KUKA KRL program: Milling_8_2.src

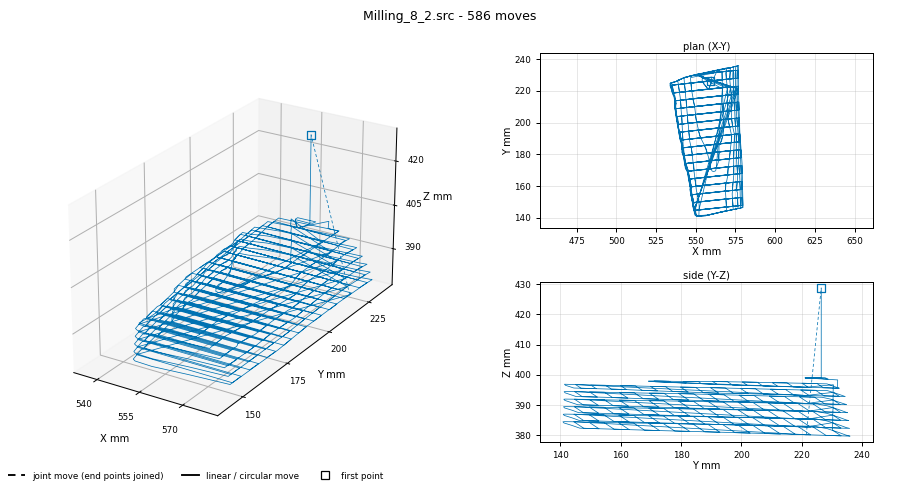
[picture p0: tool path of Milling_8_2.src, 586 of 588 moves have a stored position in this frame; points joined in program order, loops and branches not executed]
&ACCESS RVP
&REL 1
&PARAM TEMPLATE = C:\KRC\Roboter\Template\vorgabe
&PARAM EDITMASK = *
DEF Milling_8_2 ( )


;FOLD INI
;FOLD BASISTECH INI
GLOBAL INTERRUPT DECL 3 WHEN $STOPMESS==TRUE DO IR_STOPM ( )
INTERRUPT ON 3
BAS (#INITMOV,0 )
;ENDFOLD (BASISTECH INI)
;ENDFOLD (INI)

;FOLD STARTPOSITION - BASE IS 0, TOOL IS 5, SPEED IS 15%, POSITION IS A1 5,A2 -90,A3 100,A4 5,A5 -10,A6 -5,E1 0,E2 0,E3 0,E4 0
$BWDSTART = FALSE
PDAT_ACT = {VEL 15,ACC 100,APO_DIST 50}
FDAT_ACT = {TOOL_NO 5,BASE_NO 0,IPO_FRAME #BASE}
BAS (#PTP_PARAMS,15)
PTP  {A1 5,A2 -90,A3 100,A4 5,A5 -10,A6 -5,E1 0,E2 0,E3 0,E4 0}
;ENDFOLD

;FOLD LIN SPEED IS 0.1 m/sec, INTERPOLATION SETTINGS IN FOLD
$VEL.CP=0.1
$ADVANCE=3
;ENDFOLD

BAS(#VEL_PTP,2)
PTP {X 559.273, Y 226.42, Z 428.722, A -154.581, B 85.803, C -170.798, E1 0, E2 0, E3 0, E4 0, S 'B010'}
$VEL.CP=0.012
LIN {X 559.273, Y 226.42, Z 398.722, A -154.581, B 85.803, C -170.798, E1 0, E2 0, E3 0, E4 0}
LIN {X 554.276, Y 225.886, Z 399.07, A -154.581, B 85.803, C -170.798, E1 0, E2 0, E3 0, E4 0}
LIN {X 557.594, Y 221.214, Z 398.997, A -154.581, B 85.803, C -170.798, E1 0, E2 0, E3 0, E4 0}
LIN {X 558.179, Y 221.276, Z 398.957, A -154.581, B 85.803, C -170.798, E1 0, E2 0, E3 0, E4 0}
LIN {X 558.124, Y 221.152, Z 398.964, A -154.581, B 85.803, C -170.798, E1 0, E2 0, E3 0, E4 0}
LIN {X 559.233, Y 224.054, Z 398.799, A -154.581, B 85.803, C -170.798, E1 0, E2 0, E3 0, E4 0}
LIN {X 559.279, Y 226.805, Z 398.71, A -154.581, B 85.803, C -170.798, E1 0, E2 0, E3 0, E4 0}
LIN {X 559.896, Y 227.132, Z 398.659, A -154.581, B 85.803, C -170.798, E1 0, E2 0, E3 0, E4 0}
LIN {X 560.102, Y 228.698, Z 398.595, A -154.581, B 85.803, C -170.798, E1 0, E2 0, E3 0, E4 0}
LIN {X 554.041, Y 227.675, Z 399.029, A -154.581, B 85.803, C -170.798, E1 0, E2 0, E3 0, E4 0}
LIN {X 554.023, Y 226.451, Z 399.069, A -154.581, B 85.803, C -170.798, E1 0, E2 0, E3 0, E4 0}
LIN {X 555.02, Y 224.234, Z 399.073, A -154.581, B 85.803, C -170.798, E1 0, E2 0, E3 0, E4 0}
LIN {X 557.587, Y 221.412, Z 398.992, A -154.581, B 85.803, C -170.798, E1 0, E2 0, E3 0, E4 0}
LIN {X 557.599, Y 221.063, Z 399.002, A -154.581, B 85.803, C -170.798, E1 0, E2 0, E3 0, E4 0}
LIN {X 557.929, Y 221.029, Z 398.981, A -154.581, B 85.803, C -170.798, E1 0, E2 0, E3 0, E4 0}
LIN {X 558.124, Y 221.152, Z 398.964, A -154.581, B 85.803, C -170.798, E1 0, E2 0, E3 0, E4 0}
LIN {X 563.082, Y 231.869, Z 398.3, A -154.581, B 85.803, C -170.798, E1 0, E2 0, E3 0, E4 0}
LIN {X 562.917, Y 231.79, Z 395.806, A -154.581, B 85.803, C -170.798, E1 0, E2 0, E3 0, E4 0}
LIN {X 566.518, Y 232.175, Z 395.555, A -154.581, B 85.803, C -170.798, E1 0, E2 0, E3 0, E4 0}
LIN {X 566.596, Y 227.157, Z 395.708, A -154.581, B 85.803, C -170.798, E1 0, E2 0, E3 0, E4 0}
LIN {X 546.975, Y 225.06, Z 397.075, A -154.581, B 85.803, C -170.798, E1 0, E2 0, E3 0, E4 0}
LIN {X 547.397, Y 220.078, Z 397.204, A -154.581, B 85.803, C -170.798, E1 0, E2 0, E3 0, E4 0}
LIN {X 566.723, Y 222.143, Z 395.858, A -154.581, B 85.803, C -170.798, E1 0, E2 0, E3 0, E4 0}
LIN {X 566.992, Y 217.145, Z 395.997, A -154.581, B 85.803, C -170.798, E1 0, E2 0, E3 0, E4 0}
LIN {X 548.065, Y 215.122, Z 397.316, A -154.581, B 85.803, C -170.798, E1 0, E2 0, E3 0, E4 0}
LIN {X 549.244, Y 210.221, Z 397.392, A -154.581, B 85.803, C -170.798, E1 0, E2 0, E3 0, E4 0}
LIN {X 567.155, Y 212.135, Z 396.144, A -154.581, B 85.803, C -170.798, E1 0, E2 0, E3 0, E4 0}
LIN {X 567.374, Y 207.131, Z 396.288, A -154.581, B 85.803, C -170.798, E1 0, E2 0, E3 0, E4 0}
LIN {X 549.724, Y 205.245, Z 397.517, A -154.581, B 85.803, C -170.798, E1 0, E2 0, E3 0, E4 0}
LIN {X 550.455, Y 200.296, Z 397.624, A -154.581, B 85.803, C -170.798, E1 0, E2 0, E3 0, E4 0}
LIN {X 567.339, Y 202.101, Z 396.448, A -154.581, B 85.803, C -170.798, E1 0, E2 0, E3 0, E4 0}
LIN {X 567.528, Y 197.094, Z 396.594, A -154.581, B 85.803, C -170.798, E1 0, E2 0, E3 0, E4 0}
LIN {X 551.488, Y 195.379, Z 397.711, A -154.581, B 85.803, C -170.798, E1 0, E2 0, E3 0, E4 0}
LIN {X 553.074, Y 190.522, Z 397.758, A -154.581, B 85.803, C -170.798, E1 0, E2 0, E3 0, E4 0}
LIN {X 567.026, Y 192.013, Z 396.787, A -154.581, B 85.803, C -170.798, E1 0, E2 0, E3 0, E4 0}
LIN {X 565.372, Y 186.809, Z 397.06, A -154.581, B 85.803, C -170.798, E1 0, E2 0, E3 0, E4 0}
LIN {X 555.414, Y 185.745, Z 397.754, A -154.581, B 85.803, C -170.798, E1 0, E2 0, E3 0, E4 0}
LIN {X 557.158, Y 180.904, Z 397.791, A -154.581, B 85.803, C -170.798, E1 0, E2 0, E3 0, E4 0}
LIN {X 564.666, Y 181.706, Z 397.268, A -154.581, B 85.803, C -170.798, E1 0, E2 0, E3 0, E4 0}
LIN {X 564.615, Y 176.674, Z 397.43, A -154.581, B 85.803, C -170.798, E1 0, E2 0, E3 0, E4 0}
LIN {X 558.479, Y 176.018, Z 397.857, A -154.581, B 85.803, C -170.798, E1 0, E2 0, E3 0, E4 0}
LIN {X 559.339, Y 171.083, Z 397.956, A -154.581, B 85.803, C -170.798, E1 0, E2 0, E3 0, E4 0}
LIN {X 562.949, Y 171.469, Z 397.704, A -154.581, B 85.803, C -170.798, E1 0, E2 0, E3 0, E4 0}
LIN {X 566.751, Y 221.283, Z 395.883, A -154.581, B 85.803, C -170.798, E1 0, E2 0, E3 0, E4 0}
LIN {X 566.546, Y 229.177, Z 395.648, A -154.581, B 85.803, C -170.798, E1 0, E2 0, E3 0, E4 0}
LIN {X 566.512, Y 232.489, Z 395.546, A -154.581, B 85.803, C -170.798, E1 0, E2 0, E3 0, E4 0}
LIN {X 559.172, Y 230.807, Z 396.086, A -154.581, B 85.803, C -170.798, E1 0, E2 0, E3 0, E4 0}
LIN {X 546.627, Y 228.324, Z 396.995, A -154.581, B 85.803, C -170.798, E1 0, E2 0, E3 0, E4 0}
LIN {X 547.352, Y 220.421, Z 397.196, A -154.581, B 85.803, C -170.798, E1 0, E2 0, E3 0, E4 0}
LIN {X 549.239, Y 210.57, Z 397.381, A -154.581, B 85.803, C -170.798, E1 0, E2 0, E3 0, E4 0}
LIN {X 549.237, Y 210.401, Z 397.387, A -154.581, B 85.803, C -170.798, E1 0, E2 0, E3 0, E4 0}
LIN {X 550.242, Y 201.891, Z 397.588, A -154.581, B 85.803, C -170.798, E1 0, E2 0, E3 0, E4 0}
LIN {X 552.523, Y 191.514, Z 397.764, A -154.581, B 85.803, C -170.798, E1 0, E2 0, E3 0, E4 0}
LIN {X 556.467, Y 183.635, Z 397.751, A -154.581, B 85.803, C -170.798, E1 0, E2 0, E3 0, E4 0}
LIN {X 558.139, Y 177.602, Z 397.83, A -154.581, B 85.803, C -170.798, E1 0, E2 0, E3 0, E4 0}
LIN {X 558.213, Y 176.662, Z 397.854, A -154.581, B 85.803, C -170.798, E1 0, E2 0, E3 0, E4 0}
LIN {X 558.667, Y 175.563, Z 397.859, A -154.581, B 85.803, C -170.798, E1 0, E2 0, E3 0, E4 0}
LIN {X 558.417, Y 174.065, Z 397.923, A -154.581, B 85.803, C -170.798, E1 0, E2 0, E3 0, E4 0}
LIN {X 558.896, Y 172.014, Z 397.956, A -154.581, B 85.803, C -170.798, E1 0, E2 0, E3 0, E4 0}
LIN {X 560.318, Y 169.434, Z 397.943, A -154.581, B 85.803, C -170.798, E1 0, E2 0, E3 0, E4 0}
LIN {X 561.305, Y 169.205, Z 397.884, A -154.581, B 85.803, C -170.798, E1 0, E2 0, E3 0, E4 0}
LIN {X 562.277, Y 169.501, Z 397.811, A -154.581, B 85.803, C -170.798, E1 0, E2 0, E3 0, E4 0}
LIN {X 562.575, Y 169.872, Z 397.779, A -154.581, B 85.803, C -170.798, E1 0, E2 0, E3 0, E4 0}
LIN {X 562.981, Y 171.756, Z 397.693, A -154.581, B 85.803, C -170.798, E1 0, E2 0, E3 0, E4 0}
LIN {X 564.651, Y 176.325, Z 397.438, A -154.581, B 85.803, C -170.798, E1 0, E2 0, E3 0, E4 0}
LIN {X 564.581, Y 176.991, Z 397.422, A -154.581, B 85.803, C -170.798, E1 0, E2 0, E3 0, E4 0}
LIN {X 564.319, Y 177.275, Z 397.43, A -154.581, B 85.803, C -170.798, E1 0, E2 0, E3 0, E4 0}
LIN {X 564.116, Y 178.487, Z 397.406, A -154.581, B 85.803, C -170.798, E1 0, E2 0, E3 0, E4 0}
LIN {X 564.61, Y 180.491, Z 397.31, A -154.581, B 85.803, C -170.798, E1 0, E2 0, E3 0, E4 0}
LIN {X 564.637, Y 185.466, Z 397.151, A -154.581, B 85.803, C -170.798, E1 0, E2 0, E3 0, E4 0}
LIN {X 565, Y 186.057, Z 397.109, A -154.581, B 85.803, C -170.798, E1 0, E2 0, E3 0, E4 0}
LIN {X 565.01, Y 186.246, Z 397.102, A -154.581, B 85.803, C -170.798, E1 0, E2 0, E3 0, E4 0}
LIN {X 566.215, Y 188.326, Z 396.957, A -154.581, B 85.803, C -170.798, E1 0, E2 0, E3 0, E4 0}
LIN {X 567.259, Y 192.546, Z 396.755, A -154.581, B 85.803, C -170.798, E1 0, E2 0, E3 0, E4 0}
LIN {X 567.711, Y 198.434, Z 396.539, A -154.581, B 85.803, C -170.798, E1 0, E2 0, E3 0, E4 0}
LIN {X 567.365, Y 200.775, Z 396.488, A -154.581, B 85.803, C -170.798, E1 0, E2 0, E3 0, E4 0}
LIN {X 567.009, Y 210.951, Z 396.191, A -154.581, B 85.803, C -170.798, E1 0, E2 0, E3 0, E4 0}
LIN {X 567.109, Y 211.539, Z 396.166, A -154.581, B 85.803, C -170.798, E1 0, E2 0, E3 0, E4 0}
LIN {X 566.841, Y 217.785, Z 395.987, A -154.581, B 85.803, C -170.798, E1 0, E2 0, E3 0, E4 0}
LIN {X 566.751, Y 221.283, Z 395.883, A -154.581, B 85.803, C -170.798, E1 0, E2 0, E3 0, E4 0}
LIN {X 550.024, Y 230.427, Z 396.705, A -154.581, B 85.803, C -170.798, E1 0, E2 0, E3 0, E4 0}
LIN {X 549.859, Y 230.349, Z 394.212, A -154.581, B 85.803, C -170.798, E1 0, E2 0, E3 0, E4 0}
LIN {X 569.128, Y 232.408, Z 392.87, A -154.581, B 85.803, C -170.798, E1 0, E2 0, E3 0, E4 0}
LIN {X 569.258, Y 227.395, Z 393.019, A -154.581, B 85.803, C -170.798, E1 0, E2 0, E3 0, E4 0}
LIN {X 542.858, Y 224.573, Z 394.858, A -154.581, B 85.803, C -170.798, E1 0, E2 0, E3 0, E4 0}
LIN {X 543.477, Y 219.612, Z 394.973, A -154.581, B 85.803, C -170.798, E1 0, E2 0, E3 0, E4 0}
LIN {X 569.897, Y 222.436, Z 393.133, A -154.581, B 85.803, C -170.798, E1 0, E2 0, E3 0, E4 0}
LIN {X 569.92, Y 217.411, Z 393.29, A -154.581, B 85.803, C -170.798, E1 0, E2 0, E3 0, E4 0}
LIN {X 543.976, Y 214.639, Z 395.096, A -154.581, B 85.803, C -170.798, E1 0, E2 0, E3 0, E4 0}
LIN {X 544.34, Y 209.65, Z 395.229, A -154.581, B 85.803, C -170.798, E1 0, E2 0, E3 0, E4 0}
LIN {X 570.051, Y 212.398, Z 393.439, A -154.581, B 85.803, C -170.798, E1 0, E2 0, E3 0, E4 0}
LIN {X 570.026, Y 207.369, Z 393.599, A -154.581, B 85.803, C -170.798, E1 0, E2 0, E3 0, E4 0}
LIN {X 544.695, Y 204.661, Z 395.363, A -154.581, B 85.803, C -170.798, E1 0, E2 0, E3 0, E4 0}
LIN {X 544.993, Y 199.666, Z 395.501, A -154.581, B 85.803, C -170.798, E1 0, E2 0, E3 0, E4 0}
LIN {X 570.4, Y 202.381, Z 393.731, A -154.581, B 85.803, C -170.798, E1 0, E2 0, E3 0, E4 0}
LIN {X 571.157, Y 197.435, Z 393.837, A -154.581, B 85.803, C -170.798, E1 0, E2 0, E3 0, E4 0}
LIN {X 545.573, Y 194.701, Z 395.618, A -154.581, B 85.803, C -170.798, E1 0, E2 0, E3 0, E4 0}
LIN {X 546.07, Y 189.727, Z 395.742, A -154.581, B 85.803, C -170.798, E1 0, E2 0, E3 0, E4 0}
LIN {X 572.382, Y 192.539, Z 393.91, A -154.581, B 85.803, C -170.798, E1 0, E2 0, E3 0, E4 0}
LIN {X 572.464, Y 187.521, Z 394.062, A -154.581, B 85.803, C -170.798, E1 0, E2 0, E3 0, E4 0}
LIN {X 547.032, Y 184.803, Z 395.834, A -154.581, B 85.803, C -170.798, E1 0, E2 0, E3 0, E4 0}
LIN {X 547.782, Y 179.856, Z 395.94, A -154.581, B 85.803, C -170.798, E1 0, E2 0, E3 0, E4 0}
LIN {X 571.708, Y 182.413, Z 394.273, A -154.581, B 85.803, C -170.798, E1 0, E2 0, E3 0, E4 0}
LIN {X 571.179, Y 177.329, Z 394.469, A -154.581, B 85.803, C -170.798, E1 0, E2 0, E3 0, E4 0}
LIN {X 548.499, Y 174.905, Z 396.048, A -154.581, B 85.803, C -170.798, E1 0, E2 0, E3 0, E4 0}
LIN {X 549, Y 169.932, Z 396.171, A -154.581, B 85.803, C -170.798, E1 0, E2 0, E3 0, E4 0}
LIN {X 570.412, Y 172.22, Z 394.68, A -154.581, B 85.803, C -170.798, E1 0, E2 0, E3 0, E4 0}
LIN {X 570.176, Y 167.168, Z 394.855, A -154.581, B 85.803, C -170.798, E1 0, E2 0, E3 0, E4 0}
LIN {X 549.377, Y 164.945, Z 396.304, A -154.581, B 85.803, C -170.798, E1 0, E2 0, E3 0, E4 0}
LIN {X 550.223, Y 160.008, Z 396.403, A -154.581, B 85.803, C -170.798, E1 0, E2 0, E3 0, E4 0}
LIN {X 568.972, Y 162.012, Z 395.097, A -154.581, B 85.803, C -170.798, E1 0, E2 0, E3 0, E4 0}
LIN {X 568.74, Y 156.96, Z 395.272, A -154.581, B 85.803, C -170.798, E1 0, E2 0, E3 0, E4 0}
LIN {X 550.843, Y 155.048, Z 396.518, A -154.581, B 85.803, C -170.798, E1 0, E2 0, E3 0, E4 0}
LIN {X 551.901, Y 150.134, Z 396.603, A -154.581, B 85.803, C -170.798, E1 0, E2 0, E3 0, E4 0}
LIN {X 568.944, Y 151.955, Z 395.416, A -154.581, B 85.803, C -170.798, E1 0, E2 0, E3 0, E4 0}
LIN {X 569.257, Y 146.961, Z 395.552, A -154.581, B 85.803, C -170.798, E1 0, E2 0, E3 0, E4 0}
LIN {X 552.034, Y 145.121, Z 396.752, A -154.581, B 85.803, C -170.798, E1 0, E2 0, E3 0, E4 0}
LIN {X 569.895, Y 221.552, Z 393.161, A -154.581, B 85.803, C -170.798, E1 0, E2 0, E3 0, E4 0}
LIN {X 568.905, Y 230.85, Z 392.934, A -154.581, B 85.803, C -170.798, E1 0, E2 0, E3 0, E4 0}
LIN {X 569.295, Y 233.395, Z 392.828, A -154.581, B 85.803, C -170.798, E1 0, E2 0, E3 0, E4 0}
LIN {X 569.32, Y 234.371, Z 392.795, A -154.581, B 85.803, C -170.798, E1 0, E2 0, E3 0, E4 0}
LIN {X 563.112, Y 233.1, Z 393.247, A -154.581, B 85.803, C -170.798, E1 0, E2 0, E3 0, E4 0}
LIN {X 549.519, Y 230.193, Z 394.239, A -154.581, B 85.803, C -170.798, E1 0, E2 0, E3 0, E4 0}
LIN {X 542.46, Y 228.43, Z 394.763, A -154.581, B 85.803, C -170.798, E1 0, E2 0, E3 0, E4 0}
LIN {X 542.662, Y 226.994, Z 394.794, A -154.581, B 85.803, C -170.798, E1 0, E2 0, E3 0, E4 0}
LIN {X 544.531, Y 206.697, Z 395.31, A -154.581, B 85.803, C -170.798, E1 0, E2 0, E3 0, E4 0}
LIN {X 546.184, Y 188.309, Z 395.779, A -154.581, B 85.803, C -170.798, E1 0, E2 0, E3 0, E4 0}
LIN {X 547.455, Y 182.607, Z 395.875, A -154.581, B 85.803, C -170.798, E1 0, E2 0, E3 0, E4 0}
LIN {X 548.958, Y 168.7, Z 396.213, A -154.581, B 85.803, C -170.798, E1 0, E2 0, E3 0, E4 0}
LIN {X 550.409, Y 157.059, Z 396.484, A -154.581, B 85.803, C -170.798, E1 0, E2 0, E3 0, E4 0}
LIN {X 551.877, Y 151.942, Z 396.547, A -154.581, B 85.803, C -170.798, E1 0, E2 0, E3 0, E4 0}
LIN {X 552.114, Y 147.138, Z 396.683, A -154.581, B 85.803, C -170.798, E1 0, E2 0, E3 0, E4 0}
LIN {X 551.947, Y 141.437, Z 396.874, A -154.581, B 85.803, C -170.798, E1 0, E2 0, E3 0, E4 0}
LIN {X 557.049, Y 141.764, Z 396.525, A -154.581, B 85.803, C -170.798, E1 0, E2 0, E3 0, E4 0}
LIN {X 569.361, Y 144.559, Z 395.621, A -154.581, B 85.803, C -170.798, E1 0, E2 0, E3 0, E4 0}
LIN {X 569.217, Y 148.746, Z 395.499, A -154.581, B 85.803, C -170.798, E1 0, E2 0, E3 0, E4 0}
LIN {X 568.61, Y 157.781, Z 395.255, A -154.581, B 85.803, C -170.798, E1 0, E2 0, E3 0, E4 0}
LIN {X 568.994, Y 162.281, Z 395.087, A -154.581, B 85.803, C -170.798, E1 0, E2 0, E3 0, E4 0}
LIN {X 569.458, Y 163.145, Z 395.029, A -154.581, B 85.803, C -170.798, E1 0, E2 0, E3 0, E4 0}
LIN {X 569.95, Y 165.643, Z 394.918, A -154.581, B 85.803, C -170.798, E1 0, E2 0, E3 0, E4 0}
LIN {X 570.282, Y 170.547, Z 394.742, A -154.581, B 85.803, C -170.798, E1 0, E2 0, E3 0, E4 0}
LIN {X 571.088, Y 176.308, Z 394.507, A -154.581, B 85.803, C -170.798, E1 0, E2 0, E3 0, E4 0}
LIN {X 572.666, Y 191.396, Z 393.927, A -154.581, B 85.803, C -170.798, E1 0, E2 0, E3 0, E4 0}
LIN {X 570.393, Y 201.539, Z 393.758, A -154.581, B 85.803, C -170.798, E1 0, E2 0, E3 0, E4 0}
LIN {X 570.076, Y 208.44, Z 393.562, A -154.581, B 85.803, C -170.798, E1 0, E2 0, E3 0, E4 0}
LIN {X 570.031, Y 220.272, Z 393.192, A -154.581, B 85.803, C -170.798, E1 0, E2 0, E3 0, E4 0}
LIN {X 569.895, Y 221.552, Z 393.161, A -154.581, B 85.803, C -170.798, E1 0, E2 0, E3 0, E4 0}
LIN {X 550.167, Y 230.396, Z 394.189, A -154.581, B 85.803, C -170.798, E1 0, E2 0, E3 0, E4 0}
LIN {X 550.001, Y 230.318, Z 391.696, A -154.581, B 85.803, C -170.798, E1 0, E2 0, E3 0, E4 0}
LIN {X 571.709, Y 232.638, Z 390.185, A -154.581, B 85.803, C -170.798, E1 0, E2 0, E3 0, E4 0}
LIN {X 571.367, Y 227.574, Z 390.367, A -154.581, B 85.803, C -170.798, E1 0, E2 0, E3 0, E4 0}
LIN {X 539.058, Y 224.121, Z 392.617, A -154.581, B 85.803, C -170.798, E1 0, E2 0, E3 0, E4 0}
LIN {X 539.697, Y 219.162, Z 392.731, A -154.581, B 85.803, C -170.798, E1 0, E2 0, E3 0, E4 0}
LIN {X 571.93, Y 222.607, Z 390.486, A -154.581, B 85.803, C -170.798, E1 0, E2 0, E3 0, E4 0}
LIN {X 572.421, Y 217.632, Z 390.61, A -154.581, B 85.803, C -170.798, E1 0, E2 0, E3 0, E4 0}
LIN {X 540.347, Y 214.205, Z 392.844, A -154.581, B 85.803, C -170.798, E1 0, E2 0, E3 0, E4 0}
LIN {X 540.864, Y 209.233, Z 392.966, A -154.581, B 85.803, C -170.798, E1 0, E2 0, E3 0, E4 0}
LIN {X 572.66, Y 212.631, Z 390.752, A -154.581, B 85.803, C -170.798, E1 0, E2 0, E3 0, E4 0}
LIN {X 572.569, Y 207.594, Z 390.916, A -154.581, B 85.803, C -170.798, E1 0, E2 0, E3 0, E4 0}
LIN {X 541.214, Y 204.243, Z 393.1, A -154.581, B 85.803, C -170.798, E1 0, E2 0, E3 0, E4 0}
LIN {X 541.377, Y 199.233, Z 393.247, A -154.581, B 85.803, C -170.798, E1 0, E2 0, E3 0, E4 0}
LIN {X 572.486, Y 202.558, Z 391.08, A -154.581, B 85.803, C -170.798, E1 0, E2 0, E3 0, E4 0}
LIN {X 573.286, Y 197.617, Z 391.183, A -154.581, B 85.803, C -170.798, E1 0, E2 0, E3 0, E4 0}
LIN {X 541.59, Y 194.229, Z 393.39, A -154.581, B 85.803, C -170.798, E1 0, E2 0, E3 0, E4 0}
LIN {X 541.88, Y 189.233, Z 393.528, A -154.581, B 85.803, C -170.798, E1 0, E2 0, E3 0, E4 0}
LIN {X 574.309, Y 192.699, Z 391.27, A -154.581, B 85.803, C -170.798, E1 0, E2 0, E3 0, E4 0}
LIN {X 574.463, Y 187.688, Z 391.418, A -154.581, B 85.803, C -170.798, E1 0, E2 0, E3 0, E4 0}
LIN {X 542.247, Y 184.245, Z 393.661, A -154.581, B 85.803, C -170.798, E1 0, E2 0, E3 0, E4 0}
LIN {X 542.889, Y 179.287, Z 393.775, A -154.581, B 85.803, C -170.798, E1 0, E2 0, E3 0, E4 0}
LIN {X 574.012, Y 182.613, Z 391.607, A -154.581, B 85.803, C -170.798, E1 0, E2 0, E3 0, E4 0}
LIN {X 573.866, Y 177.57, Z 391.776, A -154.581, B 85.803, C -170.798, E1 0, E2 0, E3 0, E4 0}
LIN {X 543.798, Y 174.357, Z 393.87, A -154.581, B 85.803, C -170.798, E1 0, E2 0, E3 0, E4 0}
LIN {X 545.348, Y 169.495, Z 393.92, A -154.581, B 85.803, C -170.798, E1 0, E2 0, E3 0, E4 0}
LIN {X 574.006, Y 172.558, Z 391.925, A -154.581, B 85.803, C -170.798, E1 0, E2 0, E3 0, E4 0}
LIN {X 573.905, Y 167.52, Z 392.09, A -154.581, B 85.803, C -170.798, E1 0, E2 0, E3 0, E4 0}
LIN {X 546.349, Y 164.575, Z 394.009, A -154.581, B 85.803, C -170.798, E1 0, E2 0, E3 0, E4 0}
LIN {X 547.161, Y 159.635, Z 394.111, A -154.581, B 85.803, C -170.798, E1 0, E2 0, E3 0, E4 0}
LIN {X 573.378, Y 162.437, Z 392.285, A -154.581, B 85.803, C -170.798, E1 0, E2 0, E3 0, E4 0}
LIN {X 573.016, Y 157.371, Z 392.469, A -154.581, B 85.803, C -170.798, E1 0, E2 0, E3 0, E4 0}
LIN {X 547.662, Y 154.661, Z 394.234, A -154.581, B 85.803, C -170.798, E1 0, E2 0, E3 0, E4 0}
LIN {X 548.777, Y 149.753, Z 394.315, A -154.581, B 85.803, C -170.798, E1 0, E2 0, E3 0, E4 0}
LIN {X 573.077, Y 152.35, Z 392.623, A -154.581, B 85.803, C -170.798, E1 0, E2 0, E3 0, E4 0}
LIN {X 573.474, Y 147.366, Z 392.753, A -154.581, B 85.803, C -170.798, E1 0, E2 0, E3 0, E4 0}
LIN {X 549.399, Y 144.793, Z 394.43, A -154.581, B 85.803, C -170.798, E1 0, E2 0, E3 0, E4 0}
LIN {X 571.902, Y 221.664, Z 390.517, A -154.581, B 85.803, C -170.798, E1 0, E2 0, E3 0, E4 0}
LIN {X 571.404, Y 227.212, Z 390.376, A -154.581, B 85.803, C -170.798, E1 0, E2 0, E3 0, E4 0}
LIN {X 571.706, Y 232.588, Z 390.186, A -154.581, B 85.803, C -170.798, E1 0, E2 0, E3 0, E4 0}
LIN {X 571.797, Y 234.773, Z 390.111, A -154.581, B 85.803, C -170.798, E1 0, E2 0, E3 0, E4 0}
LIN {X 570.437, Y 234.581, Z 390.208, A -154.581, B 85.803, C -170.798, E1 0, E2 0, E3 0, E4 0}
LIN {X 558.868, Y 231.914, Z 391.058, A -154.581, B 85.803, C -170.798, E1 0, E2 0, E3 0, E4 0}
LIN {X 546.71, Y 229.538, Z 391.939, A -154.581, B 85.803, C -170.798, E1 0, E2 0, E3 0, E4 0}
LIN {X 538.606, Y 226.677, Z 392.566, A -154.581, B 85.803, C -170.798, E1 0, E2 0, E3 0, E4 0}
LIN {X 540.174, Y 215.923, Z 392.801, A -154.581, B 85.803, C -170.798, E1 0, E2 0, E3 0, E4 0}
LIN {X 541.247, Y 201.41, Z 393.187, A -154.581, B 85.803, C -170.798, E1 0, E2 0, E3 0, E4 0}
LIN {X 542.303, Y 180.786, Z 393.767, A -154.581, B 85.803, C -170.798, E1 0, E2 0, E3 0, E4 0}
LIN {X 542.802, Y 179.591, Z 393.771, A -154.581, B 85.803, C -170.798, E1 0, E2 0, E3 0, E4 0}
LIN {X 544.211, Y 171.367, Z 393.937, A -154.581, B 85.803, C -170.798, E1 0, E2 0, E3 0, E4 0}
LIN {X 545.205, Y 169.954, Z 393.915, A -154.581, B 85.803, C -170.798, E1 0, E2 0, E3 0, E4 0}
LIN {X 545.249, Y 169.926, Z 393.913, A -154.581, B 85.803, C -170.798, E1 0, E2 0, E3 0, E4 0}
LIN {X 545.248, Y 169.878, Z 393.915, A -154.581, B 85.803, C -170.798, E1 0, E2 0, E3 0, E4 0}
LIN {X 547.188, Y 159.511, Z 394.113, A -154.581, B 85.803, C -170.798, E1 0, E2 0, E3 0, E4 0}
LIN {X 547.045, Y 158.056, Z 394.168, A -154.581, B 85.803, C -170.798, E1 0, E2 0, E3 0, E4 0}
LIN {X 548.509, Y 150.215, Z 394.318, A -154.581, B 85.803, C -170.798, E1 0, E2 0, E3 0, E4 0}
LIN {X 548.875, Y 149.583, Z 394.314, A -154.581, B 85.803, C -170.798, E1 0, E2 0, E3 0, E4 0}
LIN {X 548.912, Y 149.11, Z 394.326, A -154.581, B 85.803, C -170.798, E1 0, E2 0, E3 0, E4 0}
LIN {X 548.619, Y 148.849, Z 394.354, A -154.581, B 85.803, C -170.798, E1 0, E2 0, E3 0, E4 0}
LIN {X 548.614, Y 148.414, Z 394.368, A -154.581, B 85.803, C -170.798, E1 0, E2 0, E3 0, E4 0}
LIN {X 550.239, Y 142.044, Z 394.461, A -154.581, B 85.803, C -170.798, E1 0, E2 0, E3 0, E4 0}
LIN {X 550.32, Y 141.93, Z 394.459, A -154.581, B 85.803, C -170.798, E1 0, E2 0, E3 0, E4 0}
LIN {X 551.351, Y 141.33, Z 394.41, A -154.581, B 85.803, C -170.798, E1 0, E2 0, E3 0, E4 0}
LIN {X 556.967, Y 141.662, Z 394.027, A -154.581, B 85.803, C -170.798, E1 0, E2 0, E3 0, E4 0}
LIN {X 573.667, Y 145.278, Z 392.806, A -154.581, B 85.803, C -170.798, E1 0, E2 0, E3 0, E4 0}
LIN {X 573.467, Y 146.47, Z 392.782, A -154.581, B 85.803, C -170.798, E1 0, E2 0, E3 0, E4 0}
LIN {X 572.893, Y 154.908, Z 392.554, A -154.581, B 85.803, C -170.798, E1 0, E2 0, E3 0, E4 0}
LIN {X 572.923, Y 154.978, Z 392.55, A -154.581, B 85.803, C -170.798, E1 0, E2 0, E3 0, E4 0}
LIN {X 573.901, Y 166.792, Z 392.113, A -154.581, B 85.803, C -170.798, E1 0, E2 0, E3 0, E4 0}
LIN {X 573.86, Y 177.68, Z 391.773, A -154.581, B 85.803, C -170.798, E1 0, E2 0, E3 0, E4 0}
LIN {X 574.328, Y 192.585, Z 391.272, A -154.581, B 85.803, C -170.798, E1 0, E2 0, E3 0, E4 0}
LIN {X 572.937, Y 198.863, Z 391.167, A -154.581, B 85.803, C -170.798, E1 0, E2 0, E3 0, E4 0}
LIN {X 572.377, Y 205.897, Z 390.983, A -154.581, B 85.803, C -170.798, E1 0, E2 0, E3 0, E4 0}
LIN {X 572.588, Y 214.003, Z 390.713, A -154.581, B 85.803, C -170.798, E1 0, E2 0, E3 0, E4 0}
LIN {X 571.902, Y 221.664, Z 390.517, A -154.581, B 85.803, C -170.798, E1 0, E2 0, E3 0, E4 0}
LIN {X 550.346, Y 230.369, Z 391.669, A -154.581, B 85.803, C -170.798, E1 0, E2 0, E3 0, E4 0}
LIN {X 550.181, Y 230.291, Z 389.175, A -154.581, B 85.803, C -170.798, E1 0, E2 0, E3 0, E4 0}
LIN {X 573.613, Y 232.795, Z 387.543, A -154.581, B 85.803, C -170.798, E1 0, E2 0, E3 0, E4 0}
LIN {X 573.359, Y 227.741, Z 387.719, A -154.581, B 85.803, C -170.798, E1 0, E2 0, E3 0, E4 0}
LIN {X 535.133, Y 223.655, Z 390.382, A -154.581, B 85.803, C -170.798, E1 0, E2 0, E3 0, E4 0}
LIN {X 536.019, Y 218.723, Z 390.478, A -154.581, B 85.803, C -170.798, E1 0, E2 0, E3 0, E4 0}
LIN {X 573.621, Y 222.741, Z 387.86, A -154.581, B 85.803, C -170.798, E1 0, E2 0, E3 0, E4 0}
LIN {X 573.987, Y 217.753, Z 387.992, A -154.581, B 85.803, C -170.798, E1 0, E2 0, E3 0, E4 0}
LIN {X 537.263, Y 213.829, Z 390.55, A -154.581, B 85.803, C -170.798, E1 0, E2 0, E3 0, E4 0}
LIN {X 537.434, Y 208.82, Z 390.696, A -154.581, B 85.803, C -170.798, E1 0, E2 0, E3 0, E4 0}
LIN {X 574.164, Y 212.745, Z 388.138, A -154.581, B 85.803, C -170.798, E1 0, E2 0, E3 0, E4 0}
LIN {X 574.322, Y 207.735, Z 388.286, A -154.581, B 85.803, C -170.798, E1 0, E2 0, E3 0, E4 0}
LIN {X 538.265, Y 203.882, Z 390.797, A -154.581, B 85.803, C -170.798, E1 0, E2 0, E3 0, E4 0}
LIN {X 539.023, Y 198.936, Z 390.902, A -154.581, B 85.803, C -170.798, E1 0, E2 0, E3 0, E4 0}
LIN {X 574.554, Y 202.733, Z 388.428, A -154.581, B 85.803, C -170.798, E1 0, E2 0, E3 0, E4 0}
LIN {X 575.033, Y 197.757, Z 388.553, A -154.581, B 85.803, C -170.798, E1 0, E2 0, E3 0, E4 0}
LIN {X 540.019, Y 194.015, Z 390.991, A -154.581, B 85.803, C -170.798, E1 0, E2 0, E3 0, E4 0}
LIN {X 540.812, Y 189.073, Z 391.094, A -154.581, B 85.803, C -170.798, E1 0, E2 0, E3 0, E4 0}
LIN {X 575.536, Y 192.784, Z 388.676, A -154.581, B 85.803, C -170.798, E1 0, E2 0, E3 0, E4 0}
LIN {X 575.752, Y 187.78, Z 388.82, A -154.581, B 85.803, C -170.798, E1 0, E2 0, E3 0, E4 0}
LIN {X 541.75, Y 184.146, Z 391.187, A -154.581, B 85.803, C -170.798, E1 0, E2 0, E3 0, E4 0}
LIN {X 542.774, Y 179.228, Z 391.274, A -154.581, B 85.803, C -170.798, E1 0, E2 0, E3 0, E4 0}
LIN {X 575.731, Y 182.75, Z 388.979, A -154.581, B 85.803, C -170.798, E1 0, E2 0, E3 0, E4 0}
LIN {X 575.731, Y 177.723, Z 389.138, A -154.581, B 85.803, C -170.798, E1 0, E2 0, E3 0, E4 0}
LIN {X 543.686, Y 174.298, Z 391.369, A -154.581, B 85.803, C -170.798, E1 0, E2 0, E3 0, E4 0}
LIN {X 545.234, Y 169.437, Z 391.42, A -154.581, B 85.803, C -170.798, E1 0, E2 0, E3 0, E4 0}
LIN {X 576.035, Y 172.729, Z 389.275, A -154.581, B 85.803, C -170.798, E1 0, E2 0, E3 0, E4 0}
LIN {X 576.298, Y 167.73, Z 389.415, A -154.581, B 85.803, C -170.798, E1 0, E2 0, E3 0, E4 0}
LIN {X 546.243, Y 164.518, Z 391.508, A -154.581, B 85.803, C -170.798, E1 0, E2 0, E3 0, E4 0}
LIN {X 547.049, Y 159.577, Z 391.61, A -154.581, B 85.803, C -170.798, E1 0, E2 0, E3 0, E4 0}
LIN {X 575.982, Y 162.669, Z 389.595, A -154.581, B 85.803, C -170.798, E1 0, E2 0, E3 0, E4 0}
LIN {X 575.694, Y 157.611, Z 389.774, A -154.581, B 85.803, C -170.798, E1 0, E2 0, E3 0, E4 0}
LIN {X 547.553, Y 154.603, Z 391.733, A -154.581, B 85.803, C -170.798, E1 0, E2 0, E3 0, E4 0}
LIN {X 548.651, Y 149.694, Z 391.815, A -154.581, B 85.803, C -170.798, E1 0, E2 0, E3 0, E4 0}
LIN {X 576.238, Y 152.642, Z 389.894, A -154.581, B 85.803, C -170.798, E1 0, E2 0, E3 0, E4 0}
LIN {X 576.528, Y 147.646, Z 390.032, A -154.581, B 85.803, C -170.798, E1 0, E2 0, E3 0, E4 0}
LIN {X 549.282, Y 144.734, Z 391.93, A -154.581, B 85.803, C -170.798, E1 0, E2 0, E3 0, E4 0}
LIN {X 573.868, Y 221.672, Z 387.877, A -154.581, B 85.803, C -170.798, E1 0, E2 0, E3 0, E4 0}
LIN {X 573.495, Y 230.466, Z 387.625, A -154.581, B 85.803, C -170.798, E1 0, E2 0, E3 0, E4 0}
LIN {X 573.734, Y 235.118, Z 387.462, A -154.581, B 85.803, C -170.798, E1 0, E2 0, E3 0, E4 0}
LIN {X 572.791, Y 234.83, Z 387.534, A -154.581, B 85.803, C -170.798, E1 0, E2 0, E3 0, E4 0}
LIN {X 562.926, Y 232.899, Z 388.248, A -154.581, B 85.803, C -170.798, E1 0, E2 0, E3 0, E4 0}
LIN {X 549.333, Y 229.992, Z 389.241, A -154.581, B 85.803, C -170.798, E1 0, E2 0, E3 0, E4 0}
LIN {X 542.547, Y 228.324, Z 389.743, A -154.581, B 85.803, C -170.798, E1 0, E2 0, E3 0, E4 0}
LIN {X 537.459, Y 225.88, Z 390.157, A -154.581, B 85.803, C -170.798, E1 0, E2 0, E3 0, E4 0}
LIN {X 534.875, Y 225.268, Z 390.348, A -154.581, B 85.803, C -170.798, E1 0, E2 0, E3 0, E4 0}
LIN {X 535.51, Y 221.463, Z 390.426, A -154.581, B 85.803, C -170.798, E1 0, E2 0, E3 0, E4 0}
LIN {X 535.605, Y 221.3, Z 390.424, A -154.581, B 85.803, C -170.798, E1 0, E2 0, E3 0, E4 0}
LIN {X 536.458, Y 217.346, Z 390.492, A -154.581, B 85.803, C -170.798, E1 0, E2 0, E3 0, E4 0}
LIN {X 536.82, Y 216.854, Z 390.484, A -154.581, B 85.803, C -170.798, E1 0, E2 0, E3 0, E4 0}
LIN {X 537.684, Y 211.987, Z 390.58, A -154.581, B 85.803, C -170.798, E1 0, E2 0, E3 0, E4 0}
LIN {X 537.618, Y 211.901, Z 390.587, A -154.581, B 85.803, C -170.798, E1 0, E2 0, E3 0, E4 0}
LIN {X 537.311, Y 210.39, Z 390.655, A -154.581, B 85.803, C -170.798, E1 0, E2 0, E3 0, E4 0}
LIN {X 537.25, Y 210.265, Z 390.663, A -154.581, B 85.803, C -170.798, E1 0, E2 0, E3 0, E4 0}
LIN {X 537.78, Y 207.05, Z 390.729, A -154.581, B 85.803, C -170.798, E1 0, E2 0, E3 0, E4 0}
LIN {X 537.856, Y 205.308, Z 390.779, A -154.581, B 85.803, C -170.798, E1 0, E2 0, E3 0, E4 0}
LIN {X 538.643, Y 202.62, Z 390.811, A -154.581, B 85.803, C -170.798, E1 0, E2 0, E3 0, E4 0}
LIN {X 539.232, Y 196.636, Z 390.961, A -154.581, B 85.803, C -170.798, E1 0, E2 0, E3 0, E4 0}
LIN {X 539.927, Y 194.322, Z 390.988, A -154.581, B 85.803, C -170.798, E1 0, E2 0, E3 0, E4 0}
LIN {X 540.304, Y 191.854, Z 391.04, A -154.581, B 85.803, C -170.798, E1 0, E2 0, E3 0, E4 0}
LIN {X 541.806, Y 185.638, Z 391.137, A -154.581, B 85.803, C -170.798, E1 0, E2 0, E3 0, E4 0}
LIN {X 541.641, Y 184.662, Z 391.178, A -154.581, B 85.803, C -170.798, E1 0, E2 0, E3 0, E4 0}
LIN {X 542.035, Y 183.079, Z 391.202, A -154.581, B 85.803, C -170.798, E1 0, E2 0, E3 0, E4 0}
LIN {X 541.892, Y 181.446, Z 391.263, A -154.581, B 85.803, C -170.798, E1 0, E2 0, E3 0, E4 0}
LIN {X 542.698, Y 179.492, Z 391.271, A -154.581, B 85.803, C -170.798, E1 0, E2 0, E3 0, E4 0}
LIN {X 544.108, Y 171.268, Z 391.437, A -154.581, B 85.803, C -170.798, E1 0, E2 0, E3 0, E4 0}
LIN {X 545.101, Y 169.855, Z 391.415, A -154.581, B 85.803, C -170.798, E1 0, E2 0, E3 0, E4 0}
LIN {X 545.145, Y 169.826, Z 391.414, A -154.581, B 85.803, C -170.798, E1 0, E2 0, E3 0, E4 0}
LIN {X 545.145, Y 169.779, Z 391.415, A -154.581, B 85.803, C -170.798, E1 0, E2 0, E3 0, E4 0}
LIN {X 547.085, Y 159.412, Z 391.613, A -154.581, B 85.803, C -170.798, E1 0, E2 0, E3 0, E4 0}
LIN {X 546.941, Y 157.957, Z 391.668, A -154.581, B 85.803, C -170.798, E1 0, E2 0, E3 0, E4 0}
LIN {X 548.406, Y 150.116, Z 391.818, A -154.581, B 85.803, C -170.798, E1 0, E2 0, E3 0, E4 0}
LIN {X 548.772, Y 149.484, Z 391.814, A -154.581, B 85.803, C -170.798, E1 0, E2 0, E3 0, E4 0}
LIN {X 548.809, Y 149.011, Z 391.826, A -154.581, B 85.803, C -170.798, E1 0, E2 0, E3 0, E4 0}
LIN {X 548.515, Y 148.749, Z 391.854, A -154.581, B 85.803, C -170.798, E1 0, E2 0, E3 0, E4 0}
LIN {X 548.51, Y 148.315, Z 391.868, A -154.581, B 85.803, C -170.798, E1 0, E2 0, E3 0, E4 0}
LIN {X 550.136, Y 141.945, Z 391.961, A -154.581, B 85.803, C -170.798, E1 0, E2 0, E3 0, E4 0}
LIN {X 550.217, Y 141.831, Z 391.959, A -154.581, B 85.803, C -170.798, E1 0, E2 0, E3 0, E4 0}
LIN {X 551.248, Y 141.23, Z 391.91, A -154.581, B 85.803, C -170.798, E1 0, E2 0, E3 0, E4 0}
LIN {X 556.864, Y 141.562, Z 391.527, A -154.581, B 85.803, C -170.798, E1 0, E2 0, E3 0, E4 0}
LIN {X 576.539, Y 145.841, Z 390.088, A -154.581, B 85.803, C -170.798, E1 0, E2 0, E3 0, E4 0}
LIN {X 576.634, Y 146.497, Z 390.061, A -154.581, B 85.803, C -170.798, E1 0, E2 0, E3 0, E4 0}
LIN {X 576.525, Y 147.191, Z 390.047, A -154.581, B 85.803, C -170.798, E1 0, E2 0, E3 0, E4 0}
LIN {X 576.302, Y 155.583, Z 389.797, A -154.581, B 85.803, C -170.798, E1 0, E2 0, E3 0, E4 0}
LIN {X 576.015, Y 156.486, Z 389.788, A -154.581, B 85.803, C -170.798, E1 0, E2 0, E3 0, E4 0}
LIN {X 575.886, Y 156.65, Z 389.791, A -154.581, B 85.803, C -170.798, E1 0, E2 0, E3 0, E4 0}
LIN {X 575.67, Y 157.171, Z 389.789, A -154.581, B 85.803, C -170.798, E1 0, E2 0, E3 0, E4 0}
LIN {X 576.347, Y 165.594, Z 389.479, A -154.581, B 85.803, C -170.798, E1 0, E2 0, E3 0, E4 0}
LIN {X 575.738, Y 175.964, Z 389.193, A -154.581, B 85.803, C -170.798, E1 0, E2 0, E3 0, E4 0}
LIN {X 575.552, Y 185.756, Z 388.897, A -154.581, B 85.803, C -170.798, E1 0, E2 0, E3 0, E4 0}
LIN {X 575.752, Y 187.034, Z 388.843, A -154.581, B 85.803, C -170.798, E1 0, E2 0, E3 0, E4 0}
LIN {X 574.911, Y 198.533, Z 388.537, A -154.581, B 85.803, C -170.798, E1 0, E2 0, E3 0, E4 0}
LIN {X 574.187, Y 214.152, Z 388.093, A -154.581, B 85.803, C -170.798, E1 0, E2 0, E3 0, E4 0}
LIN {X 573.868, Y 221.672, Z 387.877, A -154.581, B 85.803, C -170.798, E1 0, E2 0, E3 0, E4 0}
LIN {X 550.337, Y 230.322, Z 389.164, A -154.581, B 85.803, C -170.798, E1 0, E2 0, E3 0, E4 0}
LIN {X 550.172, Y 230.243, Z 386.671, A -154.581, B 85.803, C -170.798, E1 0, E2 0, E3 0, E4 0}
LIN {X 574.988, Y 232.895, Z 384.942, A -154.581, B 85.803, C -170.798, E1 0, E2 0, E3 0, E4 0}
LIN {X 574.759, Y 227.844, Z 385.117, A -154.581, B 85.803, C -170.798, E1 0, E2 0, E3 0, E4 0}
LIN {X 534.278, Y 223.518, Z 387.936, A -154.581, B 85.803, C -170.798, E1 0, E2 0, E3 0, E4 0}
LIN {X 535.719, Y 218.645, Z 387.994, A -154.581, B 85.803, C -170.798, E1 0, E2 0, E3 0, E4 0}
LIN {X 574.898, Y 222.832, Z 385.265, A -154.581, B 85.803, C -170.798, E1 0, E2 0, E3 0, E4 0}
LIN {X 575.083, Y 217.824, Z 385.411, A -154.581, B 85.803, C -170.798, E1 0, E2 0, E3 0, E4 0}
LIN {X 537.031, Y 213.758, Z 388.061, A -154.581, B 85.803, C -170.798, E1 0, E2 0, E3 0, E4 0}
LIN {X 537.206, Y 208.749, Z 388.207, A -154.581, B 85.803, C -170.798, E1 0, E2 0, E3 0, E4 0}
LIN {X 575.252, Y 212.815, Z 385.557, A -154.581, B 85.803, C -170.798, E1 0, E2 0, E3 0, E4 0}
LIN {X 575.542, Y 207.819, Z 385.696, A -154.581, B 85.803, C -170.798, E1 0, E2 0, E3 0, E4 0}
LIN {X 538.032, Y 203.81, Z 388.308, A -154.581, B 85.803, C -170.798, E1 0, E2 0, E3 0, E4 0}
LIN {X 538.796, Y 198.865, Z 388.413, A -154.581, B 85.803, C -170.798, E1 0, E2 0, E3 0, E4 0}
LIN {X 575.897, Y 202.83, Z 385.829, A -154.581, B 85.803, C -170.798, E1 0, E2 0, E3 0, E4 0}
LIN {X 576.265, Y 197.842, Z 385.962, A -154.581, B 85.803, C -170.798, E1 0, E2 0, E3 0, E4 0}
LIN {X 539.785, Y 193.944, Z 388.502, A -154.581, B 85.803, C -170.798, E1 0, E2 0, E3 0, E4 0}
LIN {X 540.586, Y 189.002, Z 388.605, A -154.581, B 85.803, C -170.798, E1 0, E2 0, E3 0, E4 0}
LIN {X 576.625, Y 192.854, Z 386.095, A -154.581, B 85.803, C -170.798, E1 0, E2 0, E3 0, E4 0}
LIN {X 577.055, Y 187.873, Z 386.223, A -154.581, B 85.803, C -170.798, E1 0, E2 0, E3 0, E4 0}
LIN {X 541.519, Y 184.075, Z 388.698, A -154.581, B 85.803, C -170.798, E1 0, E2 0, E3 0, E4 0}
LIN {X 542.541, Y 179.157, Z 388.785, A -154.581, B 85.803, C -170.798, E1 0, E2 0, E3 0, E4 0}
LIN {X 577.041, Y 182.844, Z 386.383, A -154.581, B 85.803, C -170.798, E1 0, E2 0, E3 0, E4 0}
LIN {X 577.122, Y 177.826, Z 386.536, A -154.581, B 85.803, C -170.798, E1 0, E2 0, E3 0, E4 0}
LIN {X 543.455, Y 174.228, Z 388.88, A -154.581, B 85.803, C -170.798, E1 0, E2 0, E3 0, E4 0}
LIN {X 545.002, Y 169.366, Z 388.931, A -154.581, B 85.803, C -170.798, E1 0, E2 0, E3 0, E4 0}
LIN {X 577.195, Y 172.806, Z 386.689, A -154.581, B 85.803, C -170.798, E1 0, E2 0, E3 0, E4 0}
LIN {X 577.598, Y 167.822, Z 386.819, A -154.581, B 85.803, C -170.798, E1 0, E2 0, E3 0, E4 0}
LIN {X 546.016, Y 164.447, Z 389.018, A -154.581, B 85.803, C -170.798, E1 0, E2 0, E3 0, E4 0}
LIN {X 546.818, Y 159.506, Z 389.121, A -154.581, B 85.803, C -170.798, E1 0, E2 0, E3 0, E4 0}
LIN {X 577.724, Y 162.809, Z 386.969, A -154.581, B 85.803, C -170.798, E1 0, E2 0, E3 0, E4 0}
LIN {X 578.07, Y 157.819, Z 387.103, A -154.581, B 85.803, C -170.798, E1 0, E2 0, E3 0, E4 0}
LIN {X 547.323, Y 154.533, Z 389.244, A -154.581, B 85.803, C -170.798, E1 0, E2 0, E3 0, E4 0}
LIN {X 548.409, Y 149.622, Z 389.327, A -154.581, B 85.803, C -170.798, E1 0, E2 0, E3 0, E4 0}
LIN {X 578.131, Y 152.798, Z 387.257, A -154.581, B 85.803, C -170.798, E1 0, E2 0, E3 0, E4 0}
LIN {X 578.156, Y 147.774, Z 387.413, A -154.581, B 85.803, C -170.798, E1 0, E2 0, E3 0, E4 0}
LIN {X 549.047, Y 144.663, Z 389.441, A -154.581, B 85.803, C -170.798, E1 0, E2 0, E3 0, E4 0}
LIN {X 575.1, Y 221.634, Z 385.29, A -154.581, B 85.803, C -170.798, E1 0, E2 0, E3 0, E4 0}
LIN {X 574.819, Y 230.604, Z 385.026, A -154.581, B 85.803, C -170.798, E1 0, E2 0, E3 0, E4 0}
LIN {X 575.247, Y 235.526, Z 384.842, A -154.581, B 85.803, C -170.798, E1 0, E2 0, E3 0, E4 0}
LIN {X 572.567, Y 234.728, Z 385.045, A -154.581, B 85.803, C -170.798, E1 0, E2 0, E3 0, E4 0}
LIN {X 562.702, Y 232.797, Z 385.76, A -154.581, B 85.803, C -170.798, E1 0, E2 0, E3 0, E4 0}
LIN {X 549.109, Y 229.89, Z 386.752, A -154.581, B 85.803, C -170.798, E1 0, E2 0, E3 0, E4 0}
LIN {X 542.323, Y 228.222, Z 387.255, A -154.581, B 85.803, C -170.798, E1 0, E2 0, E3 0, E4 0}
LIN {X 537.234, Y 225.779, Z 387.669, A -154.581, B 85.803, C -170.798, E1 0, E2 0, E3 0, E4 0}
LIN {X 534.22, Y 224.977, Z 387.894, A -154.581, B 85.803, C -170.798, E1 0, E2 0, E3 0, E4 0}
LIN {X 534.162, Y 224.822, Z 387.903, A -154.581, B 85.803, C -170.798, E1 0, E2 0, E3 0, E4 0}
LIN {X 534.369, Y 222.628, Z 387.958, A -154.581, B 85.803, C -170.798, E1 0, E2 0, E3 0, E4 0}
LIN {X 535.381, Y 221.198, Z 387.936, A -154.581, B 85.803, C -170.798, E1 0, E2 0, E3 0, E4 0}
LIN {X 535.565, Y 219.063, Z 387.991, A -154.581, B 85.803, C -170.798, E1 0, E2 0, E3 0, E4 0}
LIN {X 536.234, Y 217.244, Z 388.004, A -154.581, B 85.803, C -170.798, E1 0, E2 0, E3 0, E4 0}
LIN {X 536.596, Y 216.752, Z 387.995, A -154.581, B 85.803, C -170.798, E1 0, E2 0, E3 0, E4 0}
LIN {X 537.459, Y 211.885, Z 388.091, A -154.581, B 85.803, C -170.798, E1 0, E2 0, E3 0, E4 0}
LIN {X 537.394, Y 211.8, Z 388.098, A -154.581, B 85.803, C -170.798, E1 0, E2 0, E3 0, E4 0}
LIN {X 537.087, Y 210.288, Z 388.166, A -154.581, B 85.803, C -170.798, E1 0, E2 0, E3 0, E4 0}
LIN {X 537.025, Y 210.162, Z 388.175, A -154.581, B 85.803, C -170.798, E1 0, E2 0, E3 0, E4 0}
LIN {X 537.556, Y 206.948, Z 388.241, A -154.581, B 85.803, C -170.798, E1 0, E2 0, E3 0, E4 0}
LIN {X 537.631, Y 205.206, Z 388.29, A -154.581, B 85.803, C -170.798, E1 0, E2 0, E3 0, E4 0}
LIN {X 538.418, Y 202.518, Z 388.323, A -154.581, B 85.803, C -170.798, E1 0, E2 0, E3 0, E4 0}
LIN {X 539.008, Y 196.534, Z 388.472, A -154.581, B 85.803, C -170.798, E1 0, E2 0, E3 0, E4 0}
LIN {X 539.703, Y 194.22, Z 388.499, A -154.581, B 85.803, C -170.798, E1 0, E2 0, E3 0, E4 0}
LIN {X 540.08, Y 191.753, Z 388.552, A -154.581, B 85.803, C -170.798, E1 0, E2 0, E3 0, E4 0}
LIN {X 541.582, Y 185.536, Z 388.648, A -154.581, B 85.803, C -170.798, E1 0, E2 0, E3 0, E4 0}
LIN {X 541.416, Y 184.561, Z 388.69, A -154.581, B 85.803, C -170.798, E1 0, E2 0, E3 0, E4 0}
LIN {X 541.811, Y 182.977, Z 388.714, A -154.581, B 85.803, C -170.798, E1 0, E2 0, E3 0, E4 0}
LIN {X 541.667, Y 181.344, Z 388.774, A -154.581, B 85.803, C -170.798, E1 0, E2 0, E3 0, E4 0}
LIN {X 542.474, Y 179.39, Z 388.783, A -154.581, B 85.803, C -170.798, E1 0, E2 0, E3 0, E4 0}
LIN {X 543.884, Y 171.167, Z 388.948, A -154.581, B 85.803, C -170.798, E1 0, E2 0, E3 0, E4 0}
LIN {X 544.877, Y 169.753, Z 388.927, A -154.581, B 85.803, C -170.798, E1 0, E2 0, E3 0, E4 0}
LIN {X 544.921, Y 169.724, Z 388.925, A -154.581, B 85.803, C -170.798, E1 0, E2 0, E3 0, E4 0}
LIN {X 544.92, Y 169.677, Z 388.926, A -154.581, B 85.803, C -170.798, E1 0, E2 0, E3 0, E4 0}
LIN {X 546.861, Y 159.31, Z 389.124, A -154.581, B 85.803, C -170.798, E1 0, E2 0, E3 0, E4 0}
LIN {X 546.717, Y 157.855, Z 389.18, A -154.581, B 85.803, C -170.798, E1 0, E2 0, E3 0, E4 0}
LIN {X 548.182, Y 150.014, Z 389.329, A -154.581, B 85.803, C -170.798, E1 0, E2 0, E3 0, E4 0}
LIN {X 548.548, Y 149.382, Z 389.325, A -154.581, B 85.803, C -170.798, E1 0, E2 0, E3 0, E4 0}
LIN {X 548.585, Y 148.909, Z 389.338, A -154.581, B 85.803, C -170.798, E1 0, E2 0, E3 0, E4 0}
LIN {X 548.291, Y 148.648, Z 389.365, A -154.581, B 85.803, C -170.798, E1 0, E2 0, E3 0, E4 0}
LIN {X 548.286, Y 148.213, Z 389.379, A -154.581, B 85.803, C -170.798, E1 0, E2 0, E3 0, E4 0}
LIN {X 549.911, Y 141.843, Z 389.472, A -154.581, B 85.803, C -170.798, E1 0, E2 0, E3 0, E4 0}
LIN {X 549.992, Y 141.729, Z 389.47, A -154.581, B 85.803, C -170.798, E1 0, E2 0, E3 0, E4 0}
LIN {X 551.023, Y 141.128, Z 389.421, A -154.581, B 85.803, C -170.798, E1 0, E2 0, E3 0, E4 0}
LIN {X 556.639, Y 141.46, Z 389.038, A -154.581, B 85.803, C -170.798, E1 0, E2 0, E3 0, E4 0}
LIN {X 567.493, Y 144.054, Z 388.237, A -154.581, B 85.803, C -170.798, E1 0, E2 0, E3 0, E4 0}
LIN {X 578.196, Y 146.142, Z 387.462, A -154.581, B 85.803, C -170.798, E1 0, E2 0, E3 0, E4 0}
LIN {X 578.085, Y 146.589, Z 387.456, A -154.581, B 85.803, C -170.798, E1 0, E2 0, E3 0, E4 0}
LIN {X 578.136, Y 147.091, Z 387.436, A -154.581, B 85.803, C -170.798, E1 0, E2 0, E3 0, E4 0}
LIN {X 577.763, Y 164.039, Z 386.927, A -154.581, B 85.803, C -170.798, E1 0, E2 0, E3 0, E4 0}
LIN {X 576.987, Y 174.464, Z 386.65, A -154.581, B 85.803, C -170.798, E1 0, E2 0, E3 0, E4 0}
LIN {X 577.136, Y 186.625, Z 386.257, A -154.581, B 85.803, C -170.798, E1 0, E2 0, E3 0, E4 0}
LIN {X 575.555, Y 207.067, Z 385.718, A -154.581, B 85.803, C -170.798, E1 0, E2 0, E3 0, E4 0}
LIN {X 575.1, Y 221.634, Z 385.29, A -154.581, B 85.803, C -170.798, E1 0, E2 0, E3 0, E4 0}
LIN {X 550.289, Y 230.27, Z 386.662, A -154.581, B 85.803, C -170.798, E1 0, E2 0, E3 0, E4 0}
LIN {X 550.124, Y 230.192, Z 384.169, A -154.581, B 85.803, C -170.798, E1 0, E2 0, E3 0, E4 0}
LIN {X 576.073, Y 232.965, Z 382.361, A -154.581, B 85.803, C -170.798, E1 0, E2 0, E3 0, E4 0}
LIN {X 575.907, Y 227.92, Z 382.531, A -154.581, B 85.803, C -170.798, E1 0, E2 0, E3 0, E4 0}
LIN {X 534.053, Y 223.447, Z 385.446, A -154.581, B 85.803, C -170.798, E1 0, E2 0, E3 0, E4 0}
LIN {X 535.488, Y 218.574, Z 385.505, A -154.581, B 85.803, C -170.798, E1 0, E2 0, E3 0, E4 0}
LIN {X 575.892, Y 222.892, Z 382.691, A -154.581, B 85.803, C -170.798, E1 0, E2 0, E3 0, E4 0}
LIN {X 576.11, Y 217.888, Z 382.834, A -154.581, B 85.803, C -170.798, E1 0, E2 0, E3 0, E4 0}
LIN {X 536.802, Y 213.687, Z 385.571, A -154.581, B 85.803, C -170.798, E1 0, E2 0, E3 0, E4 0}
LIN {X 536.981, Y 208.679, Z 385.717, A -154.581, B 85.803, C -170.798, E1 0, E2 0, E3 0, E4 0}
LIN {X 576.295, Y 212.881, Z 382.979, A -154.581, B 85.803, C -170.798, E1 0, E2 0, E3 0, E4 0}
LIN {X 576.573, Y 207.883, Z 383.118, A -154.581, B 85.803, C -170.798, E1 0, E2 0, E3 0, E4 0}
LIN {X 537.802, Y 203.74, Z 385.818, A -154.581, B 85.803, C -170.798, E1 0, E2 0, E3 0, E4 0}
LIN {X 538.572, Y 198.795, Z 385.923, A -154.581, B 85.803, C -170.798, E1 0, E2 0, E3 0, E4 0}
LIN {X 576.776, Y 202.878, Z 383.263, A -154.581, B 85.803, C -170.798, E1 0, E2 0, E3 0, E4 0}
LIN {X 577.095, Y 197.885, Z 383.399, A -154.581, B 85.803, C -170.798, E1 0, E2 0, E3 0, E4 0}
LIN {X 539.556, Y 193.873, Z 386.013, A -154.581, B 85.803, C -170.798, E1 0, E2 0, E3 0, E4 0}
LIN {X 540.362, Y 188.932, Z 386.115, A -154.581, B 85.803, C -170.798, E1 0, E2 0, E3 0, E4 0}
LIN {X 577.349, Y 192.885, Z 383.539, A -154.581, B 85.803, C -170.798, E1 0, E2 0, E3 0, E4 0}
LIN {X 577.744, Y 187.9, Z 383.67, A -154.581, B 85.803, C -170.798, E1 0, E2 0, E3 0, E4 0}
LIN {X 541.292, Y 184.004, Z 386.209, A -154.581, B 85.803, C -170.798, E1 0, E2 0, E3 0, E4 0}
LIN {X 542.311, Y 179.086, Z 386.296, A -154.581, B 85.803, C -170.798, E1 0, E2 0, E3 0, E4 0}
LIN {X 578.024, Y 182.903, Z 383.809, A -154.581, B 85.803, C -170.798, E1 0, E2 0, E3 0, E4 0}
LIN {X 578.209, Y 177.896, Z 383.955, A -154.581, B 85.803, C -170.798, E1 0, E2 0, E3 0, E4 0}
LIN {X 543.228, Y 174.157, Z 386.39, A -154.581, B 85.803, C -170.798, E1 0, E2 0, E3 0, E4 0}
LIN {X 544.773, Y 169.295, Z 386.441, A -154.581, B 85.803, C -170.798, E1 0, E2 0, E3 0, E4 0}
LIN {X 578.403, Y 172.889, Z 384.099, A -154.581, B 85.803, C -170.798, E1 0, E2 0, E3 0, E4 0}
LIN {X 578.568, Y 167.88, Z 384.246, A -154.581, B 85.803, C -170.798, E1 0, E2 0, E3 0, E4 0}
LIN {X 545.792, Y 164.377, Z 386.529, A -154.581, B 85.803, C -170.798, E1 0, E2 0, E3 0, E4 0}
LIN {X 546.59, Y 159.435, Z 386.632, A -154.581, B 85.803, C -170.798, E1 0, E2 0, E3 0, E4 0}
LIN {X 578.769, Y 162.874, Z 384.39, A -154.581, B 85.803, C -170.798, E1 0, E2 0, E3 0, E4 0}
LIN {X 578.911, Y 157.862, Z 384.539, A -154.581, B 85.803, C -170.798, E1 0, E2 0, E3 0, E4 0}
LIN {X 547.097, Y 154.462, Z 386.754, A -154.581, B 85.803, C -170.798, E1 0, E2 0, E3 0, E4 0}
LIN {X 548.173, Y 149.55, Z 386.838, A -154.581, B 85.803, C -170.798, E1 0, E2 0, E3 0, E4 0}
LIN {X 578.967, Y 152.841, Z 384.693, A -154.581, B 85.803, C -170.798, E1 0, E2 0, E3 0, E4 0}
LIN {X 579.135, Y 147.832, Z 384.84, A -154.581, B 85.803, C -170.798, E1 0, E2 0, E3 0, E4 0}
LIN {X 548.817, Y 144.592, Z 386.951, A -154.581, B 85.803, C -170.798, E1 0, E2 0, E3 0, E4 0}
LIN {X 575.954, Y 221.535, Z 382.729, A -154.581, B 85.803, C -170.798, E1 0, E2 0, E3 0, E4 0}
LIN {X 576.183, Y 234.38, Z 382.31, A -154.581, B 85.803, C -170.798, E1 0, E2 0, E3 0, E4 0}
LIN {X 576.333, Y 235.814, Z 382.255, A -154.581, B 85.803, C -170.798, E1 0, E2 0, E3 0, E4 0}
LIN {X 572.345, Y 234.632, Z 382.556, A -154.581, B 85.803, C -170.798, E1 0, E2 0, E3 0, E4 0}
LIN {X 562.48, Y 232.701, Z 383.271, A -154.581, B 85.803, C -170.798, E1 0, E2 0, E3 0, E4 0}
LIN {X 548.886, Y 229.794, Z 384.263, A -154.581, B 85.803, C -170.798, E1 0, E2 0, E3 0, E4 0}
LIN {X 542.1, Y 228.126, Z 384.766, A -154.581, B 85.803, C -170.798, E1 0, E2 0, E3 0, E4 0}
LIN {X 537.012, Y 225.683, Z 385.18, A -154.581, B 85.803, C -170.798, E1 0, E2 0, E3 0, E4 0}
LIN {X 533.998, Y 224.881, Z 385.405, A -154.581, B 85.803, C -170.798, E1 0, E2 0, E3 0, E4 0}
LIN {X 533.939, Y 224.726, Z 385.413, A -154.581, B 85.803, C -170.798, E1 0, E2 0, E3 0, E4 0}
LIN {X 534.147, Y 222.532, Z 385.469, A -154.581, B 85.803, C -170.798, E1 0, E2 0, E3 0, E4 0}
LIN {X 535.159, Y 221.102, Z 385.447, A -154.581, B 85.803, C -170.798, E1 0, E2 0, E3 0, E4 0}
LIN {X 535.343, Y 218.967, Z 385.502, A -154.581, B 85.803, C -170.798, E1 0, E2 0, E3 0, E4 0}
LIN {X 536.012, Y 217.148, Z 385.515, A -154.581, B 85.803, C -170.798, E1 0, E2 0, E3 0, E4 0}
LIN {X 536.374, Y 216.656, Z 385.506, A -154.581, B 85.803, C -170.798, E1 0, E2 0, E3 0, E4 0}
LIN {X 537.237, Y 211.789, Z 385.602, A -154.581, B 85.803, C -170.798, E1 0, E2 0, E3 0, E4 0}
LIN {X 537.172, Y 211.703, Z 385.609, A -154.581, B 85.803, C -170.798, E1 0, E2 0, E3 0, E4 0}
LIN {X 536.865, Y 210.192, Z 385.677, A -154.581, B 85.803, C -170.798, E1 0, E2 0, E3 0, E4 0}
LIN {X 536.803, Y 210.066, Z 385.685, A -154.581, B 85.803, C -170.798, E1 0, E2 0, E3 0, E4 0}
LIN {X 537.334, Y 206.852, Z 385.751, A -154.581, B 85.803, C -170.798, E1 0, E2 0, E3 0, E4 0}
LIN {X 537.409, Y 205.111, Z 385.801, A -154.581, B 85.803, C -170.798, E1 0, E2 0, E3 0, E4 0}
LIN {X 538.196, Y 202.422, Z 385.834, A -154.581, B 85.803, C -170.798, E1 0, E2 0, E3 0, E4 0}
LIN {X 538.786, Y 196.438, Z 385.983, A -154.581, B 85.803, C -170.798, E1 0, E2 0, E3 0, E4 0}
LIN {X 539.481, Y 194.124, Z 386.01, A -154.581, B 85.803, C -170.798, E1 0, E2 0, E3 0, E4 0}
LIN {X 539.857, Y 191.657, Z 386.063, A -154.581, B 85.803, C -170.798, E1 0, E2 0, E3 0, E4 0}
LIN {X 541.36, Y 185.44, Z 386.159, A -154.581, B 85.803, C -170.798, E1 0, E2 0, E3 0, E4 0}
LIN {X 541.194, Y 184.465, Z 386.201, A -154.581, B 85.803, C -170.798, E1 0, E2 0, E3 0, E4 0}
LIN {X 541.589, Y 182.881, Z 386.224, A -154.581, B 85.803, C -170.798, E1 0, E2 0, E3 0, E4 0}
LIN {X 541.445, Y 181.248, Z 386.285, A -154.581, B 85.803, C -170.798, E1 0, E2 0, E3 0, E4 0}
LIN {X 542.252, Y 179.294, Z 386.293, A -154.581, B 85.803, C -170.798, E1 0, E2 0, E3 0, E4 0}
LIN {X 543.661, Y 171.071, Z 386.459, A -154.581, B 85.803, C -170.798, E1 0, E2 0, E3 0, E4 0}
LIN {X 544.655, Y 169.657, Z 386.438, A -154.581, B 85.803, C -170.798, E1 0, E2 0, E3 0, E4 0}
LIN {X 544.699, Y 169.629, Z 386.436, A -154.581, B 85.803, C -170.798, E1 0, E2 0, E3 0, E4 0}
LIN {X 544.698, Y 169.581, Z 386.437, A -154.581, B 85.803, C -170.798, E1 0, E2 0, E3 0, E4 0}
LIN {X 546.638, Y 159.215, Z 386.635, A -154.581, B 85.803, C -170.798, E1 0, E2 0, E3 0, E4 0}
LIN {X 546.495, Y 157.759, Z 386.691, A -154.581, B 85.803, C -170.798, E1 0, E2 0, E3 0, E4 0}
LIN {X 547.959, Y 149.919, Z 386.84, A -154.581, B 85.803, C -170.798, E1 0, E2 0, E3 0, E4 0}
LIN {X 548.326, Y 149.286, Z 386.836, A -154.581, B 85.803, C -170.798, E1 0, E2 0, E3 0, E4 0}
LIN {X 548.363, Y 148.813, Z 386.848, A -154.581, B 85.803, C -170.798, E1 0, E2 0, E3 0, E4 0}
LIN {X 548.069, Y 148.552, Z 386.876, A -154.581, B 85.803, C -170.798, E1 0, E2 0, E3 0, E4 0}
LIN {X 548.064, Y 148.117, Z 386.89, A -154.581, B 85.803, C -170.798, E1 0, E2 0, E3 0, E4 0}
LIN {X 549.689, Y 141.747, Z 386.983, A -154.581, B 85.803, C -170.798, E1 0, E2 0, E3 0, E4 0}
LIN {X 549.77, Y 141.633, Z 386.981, A -154.581, B 85.803, C -170.798, E1 0, E2 0, E3 0, E4 0}
LIN {X 550.801, Y 141.032, Z 386.932, A -154.581, B 85.803, C -170.798, E1 0, E2 0, E3 0, E4 0}
LIN {X 556.417, Y 141.364, Z 386.549, A -154.581, B 85.803, C -170.798, E1 0, E2 0, E3 0, E4 0}
LIN {X 567.27, Y 143.958, Z 385.748, A -154.581, B 85.803, C -170.798, E1 0, E2 0, E3 0, E4 0}
LIN {X 579.227, Y 146.348, Z 384.881, A -154.581, B 85.803, C -170.798, E1 0, E2 0, E3 0, E4 0}
LIN {X 578.916, Y 158.093, Z 384.531, A -154.581, B 85.803, C -170.798, E1 0, E2 0, E3 0, E4 0}
LIN {X 578.025, Y 182.926, Z 383.808, A -154.581, B 85.803, C -170.798, E1 0, E2 0, E3 0, E4 0}
LIN {X 577.311, Y 193.317, Z 383.528, A -154.581, B 85.803, C -170.798, E1 0, E2 0, E3 0, E4 0}
LIN {X 575.943, Y 220.91, Z 382.75, A -154.581, B 85.803, C -170.798, E1 0, E2 0, E3 0, E4 0}
LIN {X 575.954, Y 221.535, Z 382.729, A -154.581, B 85.803, C -170.798, E1 0, E2 0, E3 0, E4 0}
LIN {X 550.235, Y 230.218, Z 384.16, A -154.581, B 85.803, C -170.798, E1 0, E2 0, E3 0, E4 0}
LIN {X 550.07, Y 230.14, Z 381.667, A -154.581, B 85.803, C -170.798, E1 0, E2 0, E3 0, E4 0}
LIN {X 576.895, Y 233.007, Z 379.799, A -154.581, B 85.803, C -170.798, E1 0, E2 0, E3 0, E4 0}
LIN {X 576.801, Y 227.97, Z 379.964, A -154.581, B 85.803, C -170.798, E1 0, E2 0, E3 0, E4 0}
LIN {X 533.853, Y 223.38, Z 382.955, A -154.581, B 85.803, C -170.798, E1 0, E2 0, E3 0, E4 0}
LIN {X 535.282, Y 218.505, Z 383.014, A -154.581, B 85.803, C -170.798, E1 0, E2 0, E3 0, E4 0}
LIN {X 576.798, Y 222.942, Z 380.123, A -154.581, B 85.803, C -170.798, E1 0, E2 0, E3 0, E4 0}
LIN {X 576.874, Y 217.923, Z 380.275, A -154.581, B 85.803, C -170.798, E1 0, E2 0, E3 0, E4 0}
LIN {X 536.594, Y 213.619, Z 383.081, A -154.581, B 85.803, C -170.798, E1 0, E2 0, E3 0, E4 0}
LIN {X 536.78, Y 208.611, Z 383.226, A -154.581, B 85.803, C -170.798, E1 0, E2 0, E3 0, E4 0}
LIN {X 577.184, Y 212.929, Z 380.412, A -154.581, B 85.803, C -170.798, E1 0, E2 0, E3 0, E4 0}
LIN {X 577.398, Y 207.925, Z 380.556, A -154.581, B 85.803, C -170.798, E1 0, E2 0, E3 0, E4 0}
LIN {X 537.597, Y 203.672, Z 383.327, A -154.581, B 85.803, C -170.798, E1 0, E2 0, E3 0, E4 0}
LIN {X 538.375, Y 198.728, Z 383.432, A -154.581, B 85.803, C -170.798, E1 0, E2 0, E3 0, E4 0}
LIN {X 577.503, Y 202.909, Z 380.707, A -154.581, B 85.803, C -170.798, E1 0, E2 0, E3 0, E4 0}
LIN {X 577.656, Y 197.899, Z 380.854, A -154.581, B 85.803, C -170.798, E1 0, E2 0, E3 0, E4 0}
LIN {X 539.351, Y 193.805, Z 383.522, A -154.581, B 85.803, C -170.798, E1 0, E2 0, E3 0, E4 0}
LIN {X 540.162, Y 188.864, Z 383.624, A -154.581, B 85.803, C -170.798, E1 0, E2 0, E3 0, E4 0}
LIN {X 577.857, Y 192.893, Z 380.999, A -154.581, B 85.803, C -170.798, E1 0, E2 0, E3 0, E4 0}
LIN {X 578.207, Y 187.903, Z 381.133, A -154.581, B 85.803, C -170.798, E1 0, E2 0, E3 0, E4 0}
LIN {X 541.089, Y 183.936, Z 383.717, A -154.581, B 85.803, C -170.798, E1 0, E2 0, E3 0, E4 0}
LIN {X 542.107, Y 179.018, Z 383.805, A -154.581, B 85.803, C -170.798, E1 0, E2 0, E3 0, E4 0}
LIN {X 578.496, Y 182.907, Z 381.271, A -154.581, B 85.803, C -170.798, E1 0, E2 0, E3 0, E4 0}
LIN {X 578.934, Y 177.927, Z 381.399, A -154.581, B 85.803, C -170.798, E1 0, E2 0, E3 0, E4 0}
LIN {X 543.025, Y 174.089, Z 383.899, A -154.581, B 85.803, C -170.798, E1 0, E2 0, E3 0, E4 0}
LIN {X 544.569, Y 169.227, Z 383.95, A -154.581, B 85.803, C -170.798, E1 0, E2 0, E3 0, E4 0}
LIN {X 579.136, Y 172.921, Z 381.543, A -154.581, B 85.803, C -170.798, E1 0, E2 0, E3 0, E4 0}
LIN {X 579.169, Y 167.898, Z 381.699, A -154.581, B 85.803, C -170.798, E1 0, E2 0, E3 0, E4 0}
LIN {X 545.593, Y 164.309, Z 384.037, A -154.581, B 85.803, C -170.798, E1 0, E2 0, E3 0, E4 0}
LIN {X 546.387, Y 159.367, Z 384.14, A -154.581, B 85.803, C -170.798, E1 0, E2 0, E3 0, E4 0}
LIN {X 579.282, Y 162.883, Z 381.849, A -154.581, B 85.803, C -170.798, E1 0, E2 0, E3 0, E4 0}
LIN {X 579.354, Y 157.863, Z 382.003, A -154.581, B 85.803, C -170.798, E1 0, E2 0, E3 0, E4 0}
LIN {X 546.896, Y 154.394, Z 384.263, A -154.581, B 85.803, C -170.798, E1 0, E2 0, E3 0, E4 0}
LIN {X 547.963, Y 149.481, Z 384.347, A -154.581, B 85.803, C -170.798, E1 0, E2 0, E3 0, E4 0}
LIN {X 579.498, Y 152.852, Z 382.151, A -154.581, B 85.803, C -170.798, E1 0, E2 0, E3 0, E4 0}
LIN {X 579.686, Y 147.845, Z 382.296, A -154.581, B 85.803, C -170.798, E1 0, E2 0, E3 0, E4 0}
LIN {X 548.611, Y 144.524, Z 384.46, A -154.581, B 85.803, C -170.798, E1 0, E2 0, E3 0, E4 0}
LIN {X 576.972, Y 221.464, Z 380.157, A -154.581, B 85.803, C -170.798, E1 0, E2 0, E3 0, E4 0}
LIN {X 576.881, Y 232.764, Z 379.807, A -154.581, B 85.803, C -170.798, E1 0, E2 0, E3 0, E4 0}
LIN {X 577.023, Y 235.953, Z 379.698, A -154.581, B 85.803, C -170.798, E1 0, E2 0, E3 0, E4 0}
LIN {X 576.934, Y 235.952, Z 379.704, A -154.581, B 85.803, C -170.798, E1 0, E2 0, E3 0, E4 0}
LIN {X 572.147, Y 234.543, Z 380.065, A -154.581, B 85.803, C -170.798, E1 0, E2 0, E3 0, E4 0}
LIN {X 562.282, Y 232.612, Z 380.78, A -154.581, B 85.803, C -170.798, E1 0, E2 0, E3 0, E4 0}
LIN {X 548.688, Y 229.705, Z 381.772, A -154.581, B 85.803, C -170.798, E1 0, E2 0, E3 0, E4 0}
LIN {X 543.269, Y 228.42, Z 382.172, A -154.581, B 85.803, C -170.798, E1 0, E2 0, E3 0, E4 0}
LIN {X 536.814, Y 225.594, Z 382.689, A -154.581, B 85.803, C -170.798, E1 0, E2 0, E3 0, E4 0}
LIN {X 533.8, Y 224.792, Z 382.914, A -154.581, B 85.803, C -170.798, E1 0, E2 0, E3 0, E4 0}
LIN {X 533.741, Y 224.637, Z 382.923, A -154.581, B 85.803, C -170.798, E1 0, E2 0, E3 0, E4 0}
LIN {X 533.949, Y 222.443, Z 382.978, A -154.581, B 85.803, C -170.798, E1 0, E2 0, E3 0, E4 0}
LIN {X 534.961, Y 221.013, Z 382.956, A -154.581, B 85.803, C -170.798, E1 0, E2 0, E3 0, E4 0}
LIN {X 535.145, Y 218.878, Z 383.011, A -154.581, B 85.803, C -170.798, E1 0, E2 0, E3 0, E4 0}
LIN {X 535.813, Y 217.059, Z 383.024, A -154.581, B 85.803, C -170.798, E1 0, E2 0, E3 0, E4 0}
LIN {X 536.176, Y 216.567, Z 383.015, A -154.581, B 85.803, C -170.798, E1 0, E2 0, E3 0, E4 0}
LIN {X 537.039, Y 211.7, Z 383.112, A -154.581, B 85.803, C -170.798, E1 0, E2 0, E3 0, E4 0}
LIN {X 536.973, Y 211.615, Z 383.119, A -154.581, B 85.803, C -170.798, E1 0, E2 0, E3 0, E4 0}
LIN {X 536.667, Y 210.104, Z 383.186, A -154.581, B 85.803, C -170.798, E1 0, E2 0, E3 0, E4 0}
LIN {X 536.605, Y 209.978, Z 383.195, A -154.581, B 85.803, C -170.798, E1 0, E2 0, E3 0, E4 0}
LIN {X 537.136, Y 206.763, Z 383.261, A -154.581, B 85.803, C -170.798, E1 0, E2 0, E3 0, E4 0}
LIN {X 537.211, Y 205.022, Z 383.31, A -154.581, B 85.803, C -170.798, E1 0, E2 0, E3 0, E4 0}
LIN {X 537.998, Y 202.333, Z 383.343, A -154.581, B 85.803, C -170.798, E1 0, E2 0, E3 0, E4 0}
LIN {X 539.283, Y 194.035, Z 383.519, A -154.581, B 85.803, C -170.798, E1 0, E2 0, E3 0, E4 0}
LIN {X 539.659, Y 191.568, Z 383.572, A -154.581, B 85.803, C -170.798, E1 0, E2 0, E3 0, E4 0}
LIN {X 541.161, Y 185.351, Z 383.668, A -154.581, B 85.803, C -170.798, E1 0, E2 0, E3 0, E4 0}
LIN {X 540.996, Y 184.376, Z 383.71, A -154.581, B 85.803, C -170.798, E1 0, E2 0, E3 0, E4 0}
LIN {X 541.391, Y 182.792, Z 383.734, A -154.581, B 85.803, C -170.798, E1 0, E2 0, E3 0, E4 0}
LIN {X 541.247, Y 181.159, Z 383.795, A -154.581, B 85.803, C -170.798, E1 0, E2 0, E3 0, E4 0}
LIN {X 542.054, Y 179.205, Z 383.803, A -154.581, B 85.803, C -170.798, E1 0, E2 0, E3 0, E4 0}
LIN {X 543.463, Y 170.982, Z 383.968, A -154.581, B 85.803, C -170.798, E1 0, E2 0, E3 0, E4 0}
LIN {X 544.457, Y 169.568, Z 383.947, A -154.581, B 85.803, C -170.798, E1 0, E2 0, E3 0, E4 0}
LIN {X 544.501, Y 169.54, Z 383.945, A -154.581, B 85.803, C -170.798, E1 0, E2 0, E3 0, E4 0}
LIN {X 544.5, Y 169.492, Z 383.947, A -154.581, B 85.803, C -170.798, E1 0, E2 0, E3 0, E4 0}
LIN {X 546.44, Y 159.126, Z 384.144, A -154.581, B 85.803, C -170.798, E1 0, E2 0, E3 0, E4 0}
LIN {X 546.297, Y 157.67, Z 384.2, A -154.581, B 85.803, C -170.798, E1 0, E2 0, E3 0, E4 0}
LIN {X 547.761, Y 149.829, Z 384.35, A -154.581, B 85.803, C -170.798, E1 0, E2 0, E3 0, E4 0}
LIN {X 548.127, Y 149.198, Z 384.345, A -154.581, B 85.803, C -170.798, E1 0, E2 0, E3 0, E4 0}
LIN {X 548.164, Y 148.724, Z 384.358, A -154.581, B 85.803, C -170.798, E1 0, E2 0, E3 0, E4 0}
LIN {X 547.871, Y 148.463, Z 384.385, A -154.581, B 85.803, C -170.798, E1 0, E2 0, E3 0, E4 0}
LIN {X 547.866, Y 148.028, Z 384.399, A -154.581, B 85.803, C -170.798, E1 0, E2 0, E3 0, E4 0}
LIN {X 549.491, Y 141.658, Z 384.492, A -154.581, B 85.803, C -170.798, E1 0, E2 0, E3 0, E4 0}
LIN {X 549.572, Y 141.544, Z 384.491, A -154.581, B 85.803, C -170.798, E1 0, E2 0, E3 0, E4 0}
LIN {X 550.603, Y 140.943, Z 384.441, A -154.581, B 85.803, C -170.798, E1 0, E2 0, E3 0, E4 0}
LIN {X 556.219, Y 141.276, Z 384.059, A -154.581, B 85.803, C -170.798, E1 0, E2 0, E3 0, E4 0}
LIN {X 567.072, Y 143.869, Z 383.258, A -154.581, B 85.803, C -170.798, E1 0, E2 0, E3 0, E4 0}
LIN {X 579.755, Y 146.522, Z 382.333, A -154.581, B 85.803, C -170.798, E1 0, E2 0, E3 0, E4 0}
LIN {X 579.156, Y 174.216, Z 381.501, A -154.581, B 85.803, C -170.798, E1 0, E2 0, E3 0, E4 0}
LIN {X 577.763, Y 193.978, Z 380.971, A -154.581, B 85.803, C -170.798, E1 0, E2 0, E3 0, E4 0}
LIN {X 577.023, Y 215.047, Z 380.356, A -154.581, B 85.803, C -170.798, E1 0, E2 0, E3 0, E4 0}
LIN {X 576.972, Y 221.464, Z 380.157, A -154.581, B 85.803, C -170.798, E1 0, E2 0, E3 0, E4 0}
PTP {X 559.273, Y 226.42, Z 428.722, A -154.581, B 85.803, C -170.798, E1 0, E2 0, E3 0, E4 0, S 'B010'}
PTP {A1 5, A2 -90, A3 100, A4 5, A5 -10, A6 -5, E1 0, E2 0, E3 0, E4 0} C_PTP

END
